FUNCTION_BLOCK Entity IMPLEMENTS I_Entity, I_Debug;
VAR
	_nId		: UDINT;
	_nStart		: UDINT;
	_nEnd		: UDINT;
	_nSize		: UDINT;
END_VAR

PROPERTY _AsIEntity : I_Entity
GET
_AsIEntity := THIS^;
END_GET
END_PROPERTY

PROPERTY INTERNAL _End : UDINT
GET
_End := _nEnd;
END_GET
SET
_nEnd := _End;
END_SET
END_PROPERTY

METHOD INTERNAL _SetSize
VAR_INPUT
	nSize	: UDINT;
END_VAR
_nSize := nSize;
END_METHOD

PROPERTY INTERNAL _Start : UDINT
GET
_Start := _nStart;
END_GET
SET
_nStart := _Start;
END_SET
END_PROPERTY

//FB_Init is always available implicitly and it is used primarily for initialization.
//The return value is not evaluated. For a specific influence, you can also declare the
//methods explicitly and provide additional code there with the standard initialization
//code. You can evaluate the return value.
METHOD FB_Init: BOOL
VAR_INPUT
    bInitRetains: BOOL; // TRUE: the retain variables are initialized (reset warm / reset cold)
    bInCopyCode: BOOL;  // TRUE: the instance will be copied to the copy code afterward (online change)
END_VAR
VAR
	_nResult	: Result;
END_VAR
IF IsErr(_RegEntity(THIS^, nIndex => _nId), nOut => _nResult) THEN
	DebugMsg(THIS^, Tc2_Standard.CONCAT('_RegEntity(THIS^) failed with code: ', TO_STRING(_nResult)));
END_IF
END_METHOD

METHOD Get : Result
VAR_INPUT
	nIndex	: UDINT;
END_VAR
VAR_OUTPUT
	iComp	: I_Component;
END_VAR
IF nIndex > _nSize - 1 OR_ELSE nIndex = 0 OR_ELSE _nSize = 0 THEN
	Get := None;
	RETURN;
END_IF

iComp := _Ec.comp[_nStart + nIndex].variant.iComponent;
Get := Ok;
END_METHOD

PROPERTY Id : UDINT
GET
Id := _nId;
END_GET
END_PROPERTY

PROPERTY Size : UDINT
GET
Size := _nSize;
END_GET
END_PROPERTY

END_FUNCTION_BLOCK

(* stored: Version 1.1.0.1
   POU Entity: Id {a3fc4420-1b23-490b-958c-b8e82c07e80d}, SpecialFunc None
   Folder _: Id {e8077190-5b33-4c5b-91af-7b20957542bb}
   Property _AsIEntity: Id {60fc76fa-dd40-4521-93f5-29f3a0849bcf}
   Get Get: Id {5b7b9954-87f2-4bb7-9b69-46ae3bdefa15}
   Property _End: Id {7ed5e455-fc58-494a-8dc6-0ca2573e5409}
   Get Get: Id {7db79da8-8058-4634-a09e-a01f1ca34087}
   Set Set: Id {77e2b638-de88-4a1a-b8f5-31e89a519e72}
   Method _SetSize: Id {341e7bbc-0303-483d-8f8d-69b5d7410f42}
   Property _Start: Id {5d53a0dc-b463-4cf0-bcbc-720c698356a0}
   Get Get: Id {b451cf7c-ffda-4cbd-9831-246d8bce73bb}
   Set Set: Id {7a9c4d16-2560-42af-ac22-20b3625b8918}
   Method Fb_init: Id {8a1c93fc-56bb-463c-aa1e-e5009cf51636}
   Method Get: Id {d850980f-263b-4ca3-bf68-c37b4aaa2580}
   Property Id: Id {4402c710-18d7-433c-9c5e-7e50ee140721}
   Get Get: Id {a6b229f7-6688-455d-b326-4d6e21f10657}
   Property Size: Id {14d02e17-8a75-4f2f-aafd-191cc43b5896}
   Get Get: Id {fd80484a-41ec-435a-93fd-cf4a1c9dc4b9} *)
